(* IEC 61131-3 sources: CodesysTest/alpha/export/PAM.dev/Plc Logic/Application/Motors/IStoredProgramMotor.itf, 1 file *)

(* ---- ExecuteStoredProgram.m.st ---- *)
(*#-#-#-#-#-#-#-#-#-#---Declaration---#-#-#-#-#-#-#-#-#-#-#-#-#*)

METHOD ExecuteStoredProgram
VAR_INPUT
    programNumber : INT;        //Program number to execute
END_VAR
